Yaskawa INFORM job: FMTV_HOOD_LOUVERS.JBI

/JOB
//NAME FMTV_HOOD_LOUVERS
//POS
///NPOS 46,0,0,0,0,0
///TOOL 0
///POSTYPE PULSE
///PULSE
C00000=66880,-160385,-79902,187543,-63186,-9823
C00001=48037,-115985,-64372,-97569,-73692,-80949
C00002=43756,-107174,-54992,-98823,-76336,-81256
C00003=42147,-103458,-50879,-99279,-77311,-81426
C00004=39917,-102438,-53411,-100320,-78994,-80558
C00005=41855,-101886,-52819,-99760,-77773,-80449
C00006=43418,-102210,-52160,-99194,-76710,-80639
C00007=87733,-105333,-23937,-72361,-51836,-91198
C00008=87733,-105333,-23937,-72361,-51836,-91198
C00009=89199,-105279,-23184,-71197,-51218,-91608
C00010=89521,-105750,-22249,-70456,-51299,-92123
C00011=65331,-111527,-18405,-81675,-64095,-93271
C00012=65651,-111662,-18558,-81498,-63944,-93281
C00013=56542,-112605,-19267,-86476,-68236,-93071
C00014=48827,-112705,-20268,-90755,-71878,-92741
C00015=26066,-106961,-53604,-104291,-87094,-82768
C00016=26039,-106855,-53492,-104299,-87110,-82771
C00017=26410,-106989,-54447,-104203,-86985,-82522
C00018=27853,-106235,-54594,-103771,-86210,-82152
C00019=39960,-102553,-53540,-100309,-78968,-80552
C00020=42213,-103617,-51056,-99261,-77271,-81419
C00021=48037,-115985,-64372,-97569,-73692,-80949
C00022=7759,-148745,-98022,-97569,-73692,-80949
C00023=-2546,-144434,-119813,-95782,48866,-70979
C00024=-57461,-121459,-67589,-86260,68490,-17853
C00025=-49644,-107395,-56809,-83219,73554,-18632
C00026=-47721,-103305,-52253,-82700,74737,-18437
C00027=-46026,-102137,-54279,-81788,76035,-19264
C00028=-48564,-101918,-53959,-82509,74418,-19369
C00029=-49602,-101746,-52945,-82925,73704,-19181
C00030=-93807,-104266,-25425,-110456,49032,-8275
C00031=-94073,-104437,-25653,-110601,48889,-8257
C00032=-96528,-104334,-24388,-112654,47877,-7504
C00033=-96896,-104639,-23824,-113266,47866,-7145
C00034=-80668,-110920,-19756,-106863,57357,-5618
C00035=-80739,-110948,-19790,-106905,57323,-5613
C00036=-73428,-111604,-20015,-102695,60786,-6036
C00037=-66405,-112477,-21734,-98509,64047,-6659
C00038=-32879,-106963,-54183,-78330,83787,-17039
C00039=-32929,-107122,-54352,-78345,83757,-17044
C00040=-33052,-106801,-54991,-78327,83781,-17316
C00041=-34435,-106195,-55367,-78695,83031,-17686
C00042=-46070,-102243,-54399,-81799,76007,-19271
C00043=-47872,-103638,-52628,-82740,74644,-18454
C00044=-57461,-121459,-67589,-86260,68490,-17853
C00045=-47368,-58389,-75463,-75325,82045,-91552
//INST
///DATE 2023/03/28 16:52
///ATTR SC,RW
///GROUP1 RB1
NOP
MOVJ C00000 VJ=65.00  //FROM HOLES
MOVJ C00001 VJ=65.00  //OVER LEFT
MOVL C00002 V=65.0  //UP TO LEFT
MOVL C00003 V=15.0  //INTO LEFT
MOVC C00004 V=25.0
MOVC C00005 V=25.0
MOVC C00006 V=25.0
MOVL C00007 V=25.0
MOVC C00008 V=25.0
MOVC C00009 V=25.0
MOVC C00010 V=25.0
MOVL C00011 V=25.0
MOVC C00012 V=25.0
MOVC C00013 V=25.0
MOVC C00014 V=25.0
MOVL C00015 V=25.0
MOVC C00016 V=25.0
MOVC C00017 V=25.0
MOVC C00018 V=25.0
MOVL C00019 V=25.0  //END
MOVL C00020 V=25.0  //AWAY FROM EDGE
MOVL C00021 V=65.0  //AWAY FROM PART
MOVJ C00022 VJ=65.00
MOVJ C00023 VJ=65.00
MOVJ C00024 VJ=65.00  //OVER RIGHT
MOVL C00025 V=65.0  //UP TO RIGHT
MOVL C00026 V=15.0  //INTO RIGHT
MOVC C00027 V=25.0  //UP TO EDGE
MOVC C00028 V=25.0
MOVC C00029 V=25.0
MOVL C00030 V=25.0
MOVC C00031 V=25.0
MOVC C00032 V=25.0
MOVC C00033 V=25.0
MOVL C00034 V=25.0
MOVC C00035 V=25.0
MOVC C00036 V=25.0
MOVC C00037 V=25.0
MOVL C00038 V=25.0
MOVC C00039 V=25.0
MOVC C00040 V=25.0
MOVC C00041 V=25.0
MOVL C00042 V=25.0  //END
MOVL C00043 V=65.0  //AWAY
MOVL C00044 V=65.0  //ABOVE
MOVL C00045 V=65.0  //CHANGE TO SAW
END
